                           END_REGION MQTT_COMMAND_SEND_PING
                         #MQTT_COMMAND_STATE_PING_RESP:
                           REGION WAIT_FOR_PING_RESP
                             //check watchdog status
                             IF #instTimerCommandWatchdog.Q THEN
                               #statEnableTimerCommandWatchdog := FALSE;
                               #statStatus := #ERR_MQTT_COMMAND_SEND_TIMEOUT; // Set correct status that identifies error clearly
                               #statSubfunctionStatus := #ERR_MQTT_COMMAND_SEND_TIMEOUT; // Status or return value of called FBs, FCs and system blocks
                               #statFBErrorState := #statFBState; // Set error state number for diagnostic 
                               #statErrorAutoCleared := TRUE;
                               #statMqttCommandState := #MQTT_COMMAND_STATE_NO_PROCESSING;
                             END_IF;
                             //Check PingRsp paket
                             CASE #tempMqttPingRspRcv OF
                               #NO_RESPONSE:  // Statement section case 1
                                 ;
                               #RESPONSE_GOOD:
                                 //disable watchdog
                                 #statEnableTimerCommandWatchdog := FALSE;
                                 //Go to no processing
                                 #statMqttCommandState := #MQTT_COMMAND_STATE_NO_PROCESSING;
                                 //set Status
                                 #statStatus := #STATUS_MQTT_CONNECTED;
                             END_CASE;
                           END_REGION MQTT_COMMAND_PING_RESP
                         ELSE  // Statement section ELSE
                           REGION ERROR_MULITPLE_INPUT
                             #statMqttCommandState := #MQTT_COMMAND_STATE_NO_PROCESSING; // reset back to idle
                             #statStatus := #ERR_MQTT_COMMAND_MULTIPLE_INPUT; // Set correct status that identifies error clearly
                             #statSubfunctionStatus := #ERR_MQTT_COMMAND_MULTIPLE_INPUT; // Status or return value of called FBs, FCs and system blocks
                             #statFBErrorState := #statFBState; // Set error state number for diagnostic 
                             #statErrorAutoCleared := TRUE;
                           END_REGION ERROR_MULITPLE_INPUT 
                       END_CASE;
                     END_REGION

                     REGION CHECK_PING_TIMER
                       //If no job is running check if keepalive experied
                       IF #statMqttCommandState = #MQTT_COMMAND_STATE_NO_PROCESSING
                         AND #instMqttKeepAliveTimer.Q THEN
                         //reset the timer
                         RESET_TIMER(#instMqttKeepAliveTimer);
                         //go to ping state
                         #statMqttCommandState := #MQTT_COMMAND_STATE_SEND_PING;
                       END_IF;
                     END_REGION CHECK_PING_TIMER

                     //Edge detection "publish / subscribe/unsubscribe" input
                     #statPublishOld := #tempPublish;
                     #statSubscribeOld := #tempSubscribe;
                     #statUnsubscribeOld := #tempUnsubscribe;

                     //Reset Done Bit
                     IF #statPublishOld = FALSE AND
                       #statSubscribeOld = FALSE AND
                       #statUnsubscribeOld = FALSE
                     THEN
                       #statDone := FALSE;
                     END_IF;

                   END_REGION CONNECTED

                 ELSE   // Undefined state in state machine reached
                   #statStatus := #ERR_UNDEFINED_STATE;
                   #statErrorUserCleared := TRUE;
               END_CASE;

             END_REGION MQTT_STATE_MACHINE
           END_IF;
         END_REGION FB_OPERATING_MONITOR_TCP

       #FB_STATE_TCP_RECONNECTING:
         REGION FB_STATE_TCP_RECONNECTING
           IF #tempTsendcStatus = #TSENDC_EST_OK THEN
             #statErrorAutoCleared := FALSE;
             //Monitor Connection
             #statFBState := #FB_STATE_OPERATING_MONITOR_TCP;
             // Begin MQTT Connection
             #statMqttConnectState := #MQTT_CONNECT_STATE_BUILD_PAKET;
           END_IF;
         END_REGION FB_STATE_TCP_RECONNECTING
       #FB_STATE_DISABLING: // Disabling active
         REGION DISABLING FB
           //  Disabling, e.g. closing connections, etc.
           // When disabling is complete the bit #statDisablingCompleted must be set
           // When MQTT is connected, send disconnect
           IF #statMqttConnectState = #MQTT_CONNECT_STATE_CONNECTED THEN
             IF #statTsendcReq = TRUE THEN
               //Interrupt any existing send jobs
               #statTsendcReq := FALSE;
             ELSE
               // INIT
               #statSendBufferPos := 0;
               //Build fixed Header
               //Message Type
               #statSendBuffer[#statSendBufferPos] := #MQTT_MSG_TYPE_DISCONNECT;
               #statSendBufferPos += 1;
               //Remaining Length (must be O)
               #statSendBuffer[#statSendBufferPos] := #REMAINIG_LEN_0;
               #statSendBufferPos += 1;
               //send request
               #statTsendcLen := #statSendBufferPos;
               #statTsendcReq := TRUE;
               #statMqttConnectState := #MQTT_CONNECT_STATE_DISCONNECTED;
             END_IF;
           ELSE
             //Disable TCP Connection
             #statTsendcReq := FALSE;
             #statTsendcEnable := FALSE;
             #statEnableTimerCommandWatchdog := TRUE;
           END_IF;
           // When TCP connection is closed
           IF #tempTsendcStatus = #TSENDC_DISCONNECTED THEN
             #statEnableTimerCommandWatchdog := FALSE;
             #statDisablingCompleted := TRUE;
           ELSIF #instTimerCommandWatchdog.Q THEN
             #statEnableTimerCommandWatchdog := FALSE;
             #statDisablingCompleted := TRUE;
           END_IF;
         END_REGION DISABLING FB
       ELSE // Undefined state in state machine reached
         #statStatus := #ERR_UNDEFINED_STATE;
         #statErrorUserCleared := TRUE;
     END_CASE;
   END_REGION STATE_MACHINE

   REGION OUTPUTS
     // Write outputs
     IF (#statDisablingCompleted = TRUE) THEN
       // Reset outputs if disabling completed
       #statValid := FALSE;
       #statBusy := FALSE;
       #statError := FALSE;
       #statDone := FALSE;
       #statErrorUserCleared := FALSE;
       #statErrorAutoCleared := FALSE;
       #statStatus := #STATUS_NO_CALL;
       // Reset application specific outputs
       #statRcvMsgStatus := #MSG_DECODE_STATUS_NO_NEW_MSG;
       #statRcvMsgDataLen := 0;
     ELSIF (#statErrorUserCleared = TRUE) AND (#statError = FALSE) THEN
       // Error can only be cleared by user; rising edge at enable input is needed to continue 
       #statValid := FALSE;
       #statBusy := FALSE;
       #statDone := FALSE;
       #statError := TRUE;
       // Write diagnostics
       #diagnostics.status := #statStatus;
       #diagnostics.subfunctionStatus := #statSubfunctionStatus;
       #diagnostics.stateNumber := #statFBErrorState;
       // execution aborted --> set state no processing
       #statTsendcEnable := FALSE; // Terminate Connection, no reason keep it up.
       #statFBState := #FB_STATE_NO_PROCESSING;
       #statMqttConnectState := #MQTT_CONNECT_STATE_NO_PROCESSING;
       #statMqttCommandState := #MQTT_COMMAND_STATE_NO_PROCESSING;
       #statRcvMsgDecodeState := #MSG_DECODE_STATE_NO_PROCESSING;

     ELSIF (#statErrorAutoCleared = TRUE) AND (#statError = FALSE) THEN
       // Error can be reset by FB automatically
       #statValid := FALSE;
       #statBusy := TRUE;
       #statError := TRUE;
       #statDone := FALSE;
       // Write diagnostics
       #diagnostics.status := #statStatus;
       #diagnostics.subfunctionStatus := #statSubfunctionStatus;
       #diagnostics.stateNumber := #statFBErrorState;
       // Handling of autocleared error
       CASE #statStatus OF
           //Just signal error and reset autocleared error afterwards.
         #ERR_MQTT_PAKET_ID_INVALID, #ERR_MQTT_SUBACK_FAILURE, #ERR_MQTT_CONNECT_TIMEOUT,
         #ERR_MQTT_COMMAND_SEND_TIMEOUT, #ERR_MQTT_COMMAND_MULTIPLE_INPUT, #ERR_CNT_EXCEEDS_ARRAY_DIMENSION,
         #ERR_MQTT_COMMAND_PUBLISH_TOPIC_INVALID, #ERR_QOS_INVALID, #ERR_MQTT_COMMAND_SUBSCRIBE_TOPIC_INVALID:
           #statErrorAutoCleared := FALSE;

         ELSE  // Statement section ELSE
           ;
       END_CASE;

     ELSIF (#statErrorAutoCleared = FALSE) AND (#statErrorUserCleared = FALSE) AND (#statError = TRUE) THEN
       // If autocleared error is acknowledged
       #statValid := TRUE;
       #statBusy := TRUE;
       #statError := FALSE;
       #statDone := FALSE;
       //   this line  more detailed status information is used instead of "#STATUS_SUBSEQUENT_CALL"
       CASE #statStatus OF
         #ERR_TCP_RECONNECTING, #ERR_MQTT_CONNECT_TIMEOUT:  // Reconnecting ok, start Mqtt reconnnect
           //set status
           #statStatus := #STATUS_MQTT_CONNECTING;
           //in the following status codes status stays connected. 
         #ERR_MQTT_PAKET_ID_INVALID, #ERR_MQTT_SUBACK_FAILURE, #ERR_MQTT_COMMAND_SEND_TIMEOUT,
         #ERR_MQTT_COMMAND_MULTIPLE_INPUT, #ERR_CNT_EXCEEDS_ARRAY_DIMENSION, #ERR_MQTT_COMMAND_PUBLISH_TOPIC_INVALID,
         #ERR_QOS_INVALID, #ERR_MQTT_COMMAND_SUBSCRIBE_TOPIC_INVALID:
           #statStatus := #STATUS_MQTT_CONNECTED;
         ELSE  // Statement section ELSE
           ;
       END_CASE;
     END_IF;

     // Write static values to outputs
     #valid := #statValid;
     #busy := #statBusy;
     #error := #statError;
     #status := #statStatus;
     //block sets ENO automatically:
     //ENO := TRUE;
     //Write application specific static values to outputs
     #done := #statDone;
     #receivedMsgStatus := #statRcvMsgStatus;
     #receivedMsgDataLen := #statRcvMsgDataLen;
   END_REGION OUTPUTS
END_FUNCTION_BLOCK

// folder: LMQTT/Utilities

FUNCTION "LMQTT_ConvertToUtf8" : Void   // FC6, SCL
TITLE = LMQTT_ConvertToUtf8
{ S7_Optimized_Access := 'TRUE' }
AUTHOR : SIEMENS
FAMILY : LMQTT
VERSION : 1.0
// Function to convert a WCHAR to a UTF-8 conformant byte sequence
   VAR_INPUT
      character : WChar;   // Character that shall be converted to UTF-8
   END_VAR
   VAR_OUTPUT
      convertedUtf8 : DWord;   // UTF-8 conformant byte sequence. B0 stores first Byte, B1 second and B2 third Byte. B3 is not used
      bytesUsed : USInt;   // Amount of Bytes converted. Ranges from 1 to 3.
      error : Bool;   // TRUE: An error occurred during the execution of the FC
      status : Word;   // 16#0000 - 16#7FFF: Status of the FC, 16#8000 - 16#FFFF: Error identification
   END_VAR
   VAR_TEMP
      tempStatus : Word;   // temp value for output 'status'
      tempConvertedUtf8 : DWord;   // temp value for output 'convertedUtf8'
      tempBytesUsed : USInt;   // temp value for output 'bytesUsed'
      tempCharacter : WChar;   // temp value for input 'character'
   END_VAR
   // Ret_Val : No return for this FC - see error and status output
   VAR CONSTANT
      STATUS_NO_ERROR : Word := 16#0000;   // no error status
      STATUS_EXECUTION_FINISHED : Word := 16#0000;   // Execution finished without errors
      ERR_UNDEFINED : Word := 16#8000;   // Error due to an undefined case
      USINT_NULL : USInt := 0;   // Init value with 0
      DWORD_NULL : DWord := 16#0000_0000;   // Init value with 0
      EMPTY_WCHAR : WChar := WCHAR#' ';   // Empty WChar for comparison
      BELOW_7F : Word := 16#007F;   // Upper limit for character if only one Byte used
      BELOW_7FF : Word := 16#07FF;   // Upper limit for character if two Byte used
      BELOW_MAX_FFFF : Word := 16#FFFF;   // Upper limit for character if three Byte used
      BYTE_3F : Byte := 16#3F;   // Conversion Value
      BYTE_80 : Byte := 16#80;   // Conversion Value
      BYTE_C0 : Byte := 16#C0;   // Conversion Value
      BYTE_E0 : Byte := 16#E0;   // Conversion Value
      USINT_ONE : USInt := 1;   // Const Value to assign amount of bytes used
      USINT_TWO : USInt := 2;   // Const Value to assign amount of bytes used
      USINT_THREE : USInt := 3;   // Const Value to assign amount of bytes used
   END_VAR
BEGIN
   REGION BLOCK INFO HEADER
       //=============================================================================
       // SIEMENS AG
       // (c)Copyright 2020
       //-----------------------------------------------------------------------------
       // Library:       LMQTT
       // Tested with:   CPU 1516-3 PN/DP V2.8
       // Engineering:   TIA Portal V16
       // Restrictions:  --
       // Requirements:  --
       // Functionality: Converts a single WChar Character to a valid UTF-8 encoded byte sequence and saves this to a DWord.
       //                The amount of bytes saved is stored in bytesUsed Output.
       //-----------------------------------------------------------------------------
       // Change log table:
       // Version    Date         Expert in charge         Changes applied
       // 03.00.00   01.10.2020   Siemens Online Support   First released version
       //=============================================================================
   END_REGION

   REGION INITIALISATION  
       // Initialize functionality: reset of variables, diagnostics, etc.
       #tempConvertedUtf8 := #DWORD_NULL;
       #tempBytesUsed := #USINT_NULL;
       #tempStatus := #STATUS_NO_ERROR;
       //assign temp value from input:
        #tempCharacter := #character;

   END_REGION

   REGION PROGRAM LOGIC
       // Use this region for application specific code
       IF #tempCharacter = #EMPTY_WCHAR THEN
           //will be only 1 byte occupied
           #tempConvertedUtf8 := WCHAR_TO_DWORD(#tempCharacter);
           #tempBytesUsed := #USINT_ONE;
       ELSIF (WCHAR_TO_WORD(#tempCharacter) <= (#BELOW_7F)) THEN
           //will be only 1 byte occupied
           #tempConvertedUtf8 := WCHAR_TO_DWORD(#tempCharacter);
           #tempBytesUsed := #USINT_ONE;
       ELSIF (WCHAR_TO_WORD(#tempCharacter) <= (#BELOW_7FF)) THEN
           //will be 2 byte occupied
           #tempConvertedUtf8.%B1 := (WCHAR_TO_BYTE(#tempCharacter) AND #BYTE_3F) OR #BYTE_80;
           #tempConvertedUtf8.%B0 := WORD_TO_BYTE(SHR(IN := WCHAR_TO_WORD(#tempCharacter), N := 6)) OR #BYTE_C0;
           #tempBytesUsed := #USINT_TWO;
       ELSIF (WCHAR_TO_WORD(#tempCharacter) <= (#BELOW_MAX_FFFF)) THEN
           //will be 3 byte occupied
           #tempConvertedUtf8.%B2 := (WCHAR_TO_BYTE(#tempCharacter) AND #BYTE_3F) OR #BYTE_80;
           #tempConvertedUtf8.%B1 := (WORD_TO_BYTE(SHR(IN := WCHAR_TO_WORD(#tempCharacter), N := 6)) AND #BYTE_3F) OR #BYTE_80;
           #tempConvertedUtf8.%B0 := WORD_TO_BYTE(SHR(IN := WCHAR_TO_WORD(#tempCharacter), N := 12)) OR #BYTE_E0;
           #tempBytesUsed := #USINT_THREE;
       END_IF;
   END_REGION

   REGION OUTPUTS
       // Write application specific temp values to outputs
       #bytesUsed := #tempBytesUsed;
       #convertedUtf8 := #tempConvertedUtf8;
       // Write error and status
       #error := #tempStatus.%X15;
       #status := #tempStatus;
       // ENO mechanism is not used --> ENO := TRUE;
       ENO := TRUE;
   END_REGION
END_FUNCTION

// ===== library types =====

FUNCTION_BLOCK "LMqtt_Publisher"   // FB2, SCL
{ S7_Optimized_Access := 'TRUE' }
VERSION : 0.1
   VAR_INPUT
      enable : Bool;
      publish : Bool;
      tcpConnParam : "typeTcpConnParam";
      mqttParam : "typeMqttParam";
   END_VAR
   VAR_OUTPUT
      tcpEstablished : Bool;
      mqttEstablished : Bool;
      published : Bool;
      busy : Bool;
      error : Bool;
      status : DWord;
      statusID : Int;
   END_VAR
   VAR
      statTcpConnParam : TCON_IP_v4;
      instTcpConnect : TCON;
      instTcpSend : TSEND;
      instTcpRCV : TRCV;
      instTcpDisconnect : TDISCON;
      instWatchDog : TON_TIME;
      instKeepAlive : TON_TIME;
      statStateMQTT : Int;
      statStateMQTTinternal : Int;
      statStateTCP : Int;
      statLastState : Int;
      statConnectLenght : Int;
      statCorrectOffset : Int;
      statSendLenght : Int;
      statConnectEncodedLenght : Int;
      statConnectLenghtOffset : Int;
      statKeepAliveTime : Time;
      statI : Int;
      statPacketID : Word;
      statPacketIDAck : Word;
      statRcvLen : UDInt;
      statPublishOld : Bool;
      statReConnect : Bool;
      statEnableOld : Bool;
      statMqttResetOld : Bool;
      statTriggerWatchDog : Bool;
      statTriggerKeepAlive : Bool;
      statNewDataRcv : Bool;
      statKeepAliveOff : Bool;
      statSendBuffer : Array[1..1000] of Byte;
      statRcvBuffer : Array[1..200] of Byte;
   END_VAR
   VAR_TEMP
      tempStringToChar : Array[0..255] of Char;
      tempCountChars : UInt;
      tempLenght : Word;
   END_VAR
   VAR CONSTANT
      TCP_PARAM : Int := 1;
      TCP_DISCONNECT : Int := -1;
      TCP_ERROR : Int := -2;
      TCP_CONNECTED : Int := 3;
      TCP_CONNECTING : Int := 2;
      MQTT_CONNECT_FLAG_CHECK : Int := 10;
      MQTT_CONNECT : Int := 11;
      MQTT_PUBLISH : Int := 13;
      MQTT_DISCONNECT : Int := 15;
      MQTT_CONNACK : Int := 12;
      MQTT_PUBACK : Int := 14;
      MQTT_PING : Int := 17;
      MQTT_PINGRESP : Int := 18;
      MQTT_PUBREL : Int := 19;
      MQTT_PUBCOMP : Int := 20;
      MQTT_IDLE : Int;
      MQTT_CONNECTED : Int := 16;
      MQTT_DISCONNECTED : Int := -11;
      MQTT_ERROR : Int := -12;
      IDLE : Int;
      TIME_MONITORING : Int := 20;
      WATCHDOG_TIME : Time := t#30s;
      MQTT_MSG_TYPE_CONNACK : Int := 32;
      MQTT_MSG_TYPE_DISCONNECT : Int := 224;
      MQTT_MSG_TYPE_PUBACK : Int := 64;
      MQTT_MSG_TYPE_PUBREC : Int := 80;
      MQTT_MSG_TYPE_PUBCOM : Int := 112;
      MQTT_MSG_TYPE_PING : Int := 192;
      MQTT_MSG_TYPE_PINGRESP : Int := 208;
      MQTT_CONNACK_ACCEPTED : Int;
      MQTT_PORT : Word := 16#22B3;
      MQTT_PROTOCOL_NAME : String := 'MQTT';
      MQTT_ERROR_WILL_FLAG : Word := 16#80F0;
      MQTT_ERROR_QOS_FLAG : Word := 16#80F1;
      MQTT_ERROR_PACKETID : Word := 16#80F2;
      MQTT_ERROR_KEEPALIVE : Word := 16#80F3;
   END_VAR
   // statTcpConnParam.ActiveEstablished := true;
BEGIN
   //=============================================================================
   //SIEMENES AG
   //(c)Copyright 2016 All Rights Reserved
   //-----------------------------------------------------------------------------
   //Library:       (that the source is dedicated to)
   //Tested with:   (target system with FW Version)
   //Engineering:   TIA Portal V15
   //Restrictions:  (OB types, etc.)
   //Requirements:  (hardware, technological package, memory needed, etc.)
   //Functionality: MQTT
   //-----------------------------------------------------------------------------
   //Change log table:
   //Version  Date       Expert in charge Changes applied
   //01.00.00 dd.mm.yyyy (name of expert) First released version
   //=============================================================================
   //Establish TCP Connection to be ready for MQTT

   IF #enable
       AND NOT #statEnableOld
   THEN
       #statStateTCP := #TCP_PARAM;
       #statStateMQTT := #MQTT_DISCONNECTED;
       #instWatchDog.IN := false;
       #statPublishOld := #publish;
       #error := 0;
       #status := 0;
       #statusID := 0;
   END_IF;

   IF NOT #enable
       AND #statEnableOld
   THEN
       IF #statStateTCP = #TCP_CONNECTED AND
           #statStateMQTT = #MQTT_DISCONNECTED
       THEN
           #statStateTCP := #TCP_DISCONNECT;
       END_IF;
       IF #statStateTCP = #TCP_CONNECTED AND
           #statStateMQTT <> #MQTT_DISCONNECTED
       THEN
           #statStateMQTT := #MQTT_DISCONNECT;
       END_IF;
       IF #statStateTCP = #TCP_CONNECTING
           OR  #statStateTCP = #IDLE
       THEN

           #statStateMQTT := #MQTT_DISCONNECTED;
           #statStateTCP := #IDLE;
       END_IF;
   END_IF;

    #instWatchDog(IN := #statTriggerWatchDog,PT := #WATCHDOG_TIME);

   REGION State maschine TCP
       CASE #statStateTCP OF
           #IDLE:
               IF NOT #error
               THEN
                   #status := 0;
                   #statusID := 0;

               END_IF;
               #statTcpConnParam.ID := #tcpConnParam.connectionID;
               #instTcpDisconnect(ID := #statTcpConnParam.ID);
               #instTcpConnect(ID := #statTcpConnParam.ID,
                               CONNECT := #statTcpConnParam);
               #published := 0;
               #busy := false;
               #mqttEstablished := false;
               #statMqttResetOld := 0;
               #tcpEstablished := false;
               #statStateMQTT := #MQTT_DISCONNECTED;
               #statStateMQTTinternal := #IDLE;
               #statTriggerWatchDog := false;
               #statTriggerKeepAlive := 0;
               IF #statLastState=#TCP_DISCONNECT
               THEN
                   #error := 0;
                   END_IF;
           #TCP_CONNECTED:
               ;
               //Check TCP Connection
               IF #instTcpRCV.STATUS > w#16#80C0
               THEN
                   #statStateTCP := #TCP_ERROR;
                   #statusID := #TCP_CONNECTED;
               END_IF;
               #statLastState := #TCP_CONNECTED;
           #TCP_PARAM:
               #statTcpConnParam.InterfaceId := #tcpConnParam.hwIdentifier;
               #statTcpConnParam.ID := #tcpConnParam.connectionID;
               #statTcpConnParam.LocalPort := #tcpConnParam.localPort;
               #statTcpConnParam.RemotePort := #tcpConnParam.mqttPort;
               #statTcpConnParam.ActiveEstablished := true;
               #statTcpConnParam.RemoteAddress.ADDR[1] := #tcpConnParam.ipAdressBroker[0];
               #statTcpConnParam.RemoteAddress.ADDR[2] := #tcpConnParam.ipAdressBroker[1];
               #statTcpConnParam.RemoteAddress.ADDR[3] := #tcpConnParam.ipAdressBroker[2];
               #statTcpConnParam.RemoteAddress.ADDR[4] := #tcpConnParam.ipAdressBroker[3];

             #statStateTCP := #TCP_CONNECTING;
           #TCP_CONNECTING:
               REGION TCP Connect
                   #statTriggerWatchDog := true;
                   #instTcpConnect.REQ := NOT #instTcpConnect.REQ XOR #instTcpConnect.BUSY;
                   #instTcpConnect(ID := #statTcpConnParam.ID,
                                   CONNECT := #statTcpConnParam);

                   IF (#instTcpConnect.DONE)
                       AND (#instTcpConnect.BUSY = 0)
                       AND (#instTcpConnect.REQ)
                   THEN
                       #instTcpConnect.REQ := false;
                       #tcpEstablished := true;
                       #statStateTCP := #TCP_CONNECTED;
                       #statTriggerWatchDog := false;
                   ELSIF (#instTcpConnect.ERROR)
                   THEN
                       #statusID := #TCP_CONNECTING;
                       #instTcpConnect.REQ := false;
                       #statStateTCP := #TCP_ERROR;
                   END_IF;
               END_REGION

           #TCP_DISCONNECT:
               REGION TCP Disconnect
                   #instTcpDisconnect.REQ := NOT #instTcpDisconnect.REQ XOR #instTcpDisconnect.BUSY;
                   #statTriggerWatchDog := false;
                   #instTcpDisconnect(ID := #statTcpConnParam.ID);

                   IF (#instTcpDisconnect.DONE)
                   THEN
                       //Done with success
                       #instTcpDisconnect.REQ := false;
                       #statLastState := #TCP_DISCONNECT;
                       #statStateTCP := #IDLE;
                   ELSIF (#instTcpDisconnect.ERROR)
                   THEN
                       #statusID := #TCP_DISCONNECT;
                       #instTcpDisconnect.REQ := false;
                       #statStateTCP := #TCP_ERROR;
                   END_IF;
               END_REGION
               ;
           #TCP_ERROR:
               REGION Errorhandling
                   #error := true;
                   #statStateMQTT := #MQTT_DISCONNECTED;
                   #statStateMQTTinternal := #IDLE;
                   #tcpEstablished := false;
                   #mqttEstablished := false;
                   #published := false;
                   #statTriggerWatchDog := false;
                   #instTcpConnect.REQ := false;
                       CASE #statusID OF
                           #TCP_CONNECTING:
                               #statStateTCP := #IDLE;
                               #status := #instTcpConnect.STATUS;
                           #TCP_CONNECTED:
                               #statStateTCP := #TCP_DISCONNECT;
                               #status := #instTcpRCV.STATUS;
                           #TCP_DISCONNECT:
                               //pointless for a retry at TDISCON
                               #statStateTCP := #IDLE;
                               #status := #instTcpDisconnect.STATUS;
                           #TIME_MONITORING:
                               IF (#statLastState = #TCP_CONNECTED)
                               THEN
                                   #statStateTCP := #TCP_DISCONNECT;
                                   #status := #instTcpRCV.STATUS;
                               ELSE
                                   #statStateTCP := #IDLE;
                                   #status := #instTcpConnect.STATUS;
                               END_IF;
                           ELSE
                               ;
                       END_CASE;
               END_REGION
               ;
           ELSE
               ;
       END_CASE;
   END_REGION
   #statEnableOld := #enable;
   REGION WatchDog
       IF #instWatchDog.Q = true
       THEN
           #statStateTCP := #TCP_ERROR;
           #statusID := #TIME_MONITORING;
       END_IF;
   END_REGION

   REGION OUC blocks

       #instTcpSend(ID:=#statTcpConnParam.ID,
                     DATA:=#statSendBuffer);
        #instTcpRCV(EN_R:=true,
                    ID:=#statTcpConnParam.ID,
                   LEN:=0,
                   ADHOC:=1,
                   RCVD_LEN=>#statRcvLen,
                   DATA:=#statRcvBuffer);
       IF #instTcpRCV.RCVD_LEN > 0 THEN
           #statNewDataRcv := 1;
       END_IF;

   END_REGION

   //Bring Statemachine in a definded state, if TCP Connection breaks
   IF #statStateMQTT > 0 AND
       #statStateTCP <> #TCP_CONNECTED
   THEN
       #statStateMQTT := #MQTT_DISCONNECTED;
       #instTcpSend.REQ := 0;
   END_IF;

   //MQTT makes no sense without an established TCP
   IF NOT (#statStateTCP = #TCP_CONNECTED)
   THEN
       RETURN;
   END_IF;




    #instKeepAlive(IN := #statTriggerKeepAlive,
                   PT := #statKeepAliveTime);
       CASE #statStateMQTT OF
           #MQTT_DISCONNECTED:
               #mqttEstablished := false;
               #statPublishOld := #publish;
               #statStateMQTT := #MQTT_CONNECT_FLAG_CHECK;
               #statStateMQTTinternal := #IDLE;
               #statTriggerKeepAlive := 0;
               #statKeepAliveOff := false;
               #statPacketID := #mqttParam.packetIdentifier;

           #MQTT_CONNECT_FLAG_CHECK:
               #busy := 1;
               //validate flags
               IF #mqttParam.connectFlag.willRetain
                   AND NOT #mqttParam.connectFlag.will
               THEN
                   #statStateMQTT := #MQTT_ERROR;
                   #statusID := #MQTT_CONNECT_FLAG_CHECK;
                   #status := #MQTT_ERROR_WILL_FLAG;
               ELSE
                   IF NOT #mqttParam.connectFlag.will
                       AND (#mqttParam.connectFlag.willQoS_1 OR #mqttParam.connectFlag.willQoS_2)
                   THEN
                       #statStateMQTT := #MQTT_ERROR;
                       #statusID := #MQTT_CONNECT_FLAG_CHECK;
                       #status := #MQTT_ERROR_QOS_FLAG;
                   ELSE
                       IF (#mqttParam.connectFlag.willQoS_1
                           AND #mqttParam.connectFlag.willQoS_2)
                       THEN
                           #statStateMQTT := #MQTT_ERROR;
                           #statusID := #MQTT_CONNECT_FLAG_CHECK;
                           #status := #MQTT_ERROR_QOS_FLAG;
                       ELSE;
                        #statStateMQTT := #MQTT_CONNECT;
                       END_IF;
                   END_IF;

               END_IF;
               IF (WORD_TO_INT(#mqttParam.keepAlive) = 0)
               THEN
                   #statKeepAliveOff := true;
               END_IF;
               IF (WORD_TO_INT(#mqttParam.keepAlive) < 2)
                   AND
                   (WORD_TO_INT(#mqttParam.keepAlive) > 0)
               THEN
                   #statStateMQTT := #MQTT_ERROR;
                   #statusID := #MQTT_CONNECT_FLAG_CHECK;
                   #status := #MQTT_ERROR_KEEPALIVE;
               END_IF;
               IF (WORD_TO_INT(#mqttParam.keepAlive) > 2)
               THEN
                   #statKeepAliveOff := false;
               END_IF;
           #MQTT_CONNECT:
                REGION MQTT Connect

                   //Calculate Remaining Lenght
                   #statConnectLenght := 10 + LEN(IN := #mqttParam.clientIdentifier) + 2;
                   IF #mqttParam.connectFlag.userName
                   THEN
                       #statConnectLenght := #statConnectLenght + LEN(IN := #mqttParam.userName) + 2;
                   END_IF;
                   IF #mqttParam.connectFlag.password
                   THEN
                       #statConnectLenght := #statConnectLenght + LEN(IN := #mqttParam.password) + 2;
                   END_IF;
                   IF #mqttParam.connectFlag.will
                   THEN
                       #statConnectLenght := #statConnectLenght + LEN(IN := #mqttParam.willMessage) + LEN(IN := #mqttParam.willTopic) + 4;
                   END_IF;
                   #statConnectLenghtOffset := 0;
                   //Build Telegram
                   //Fixed Header
                   #statSendBuffer[1] := 16#10;

                   #statSendLenght :=#statConnectLenght;
                   WHILE (#statConnectLenght > 0)
                   DO
                       #statConnectEncodedLenght := #statConnectLenght MOD 128;
                       #statConnectLenght := #statConnectLenght / 128;
                       // if there are more data to encode, set the top bit of this byte
                       IF #statConnectLenght > 0
                       THEN
                           #statConnectEncodedLenght := #statConnectEncodedLenght OR 128;
                           #statSendBuffer[2 + #statConnectLenghtOffset] := INT_TO_BYTE(#statConnectEncodedLenght);
                           #statConnectLenghtOffset := #statConnectLenghtOffset + 1;
                       ELSE
                           #statSendBuffer[2 + #statConnectLenghtOffset] := INT_TO_BYTE(#statConnectEncodedLenght);
                       END_IF;
                   END_WHILE;
                   #statSendLenght := #statSendLenght + #statConnectLenghtOffset;
                   //Variable Header
                   //Protocol name
                   #statSendBuffer[3 + #statConnectLenghtOffset] := 0;
                   #statSendBuffer[4 + #statConnectLenghtOffset] := 4;
                   #statSendBuffer[5 + #statConnectLenghtOffset] := 'M';
                   #statSendBuffer[6 + #statConnectLenghtOffset] := 'Q';
                   #statSendBuffer[7 + #statConnectLenghtOffset] := 'T';
                   #statSendBuffer[8 + #statConnectLenghtOffset] := 'T';
                   //Protocol Level
                   #statSendBuffer[9 + #statConnectLenghtOffset] := 4;
                   //Connect Flags
                   #statSendBuffer[10 + #statConnectLenghtOffset].%X0 := 0;
                   #statSendBuffer[10 + #statConnectLenghtOffset].%X1 := #mqttParam.connectFlag.cleanSession;
                   #statSendBuffer[10 + #statConnectLenghtOffset].%X2 := #mqttParam.connectFlag.will;
                   #statSendBuffer[10 + #statConnectLenghtOffset].%X3 := #mqttParam.connectFlag.willQoS_1;
                   #statSendBuffer[10 + #statConnectLenghtOffset].%X4 := #mqttParam.connectFlag.willQoS_2;
                   #statSendBuffer[10 + #statConnectLenghtOffset].%X5 := #mqttParam.connectFlag.willRetain;
                   #statSendBuffer[10 + #statConnectLenghtOffset].%X6 := #mqttParam.connectFlag.password;
                   #statSendBuffer[10 + #statConnectLenghtOffset].%X7 := #mqttParam.connectFlag.userName;
                   //Keep Alive in sec
                  #statSendBuffer[11 + #statConnectLenghtOffset] := #mqttParam.keepAlive.%B1;
                  #statSendBuffer[12 + #statConnectLenghtOffset] := #mqttParam.keepAlive.%B0;
                   //Payload
                   //ClientIdentifier
                   #tempLenght := INT_TO_WORD(LEN(IN := #mqttParam.clientIdentifier));
                   #statSendBuffer[13 + #statConnectLenghtOffset] := #tempLenght.%B1;
                   #statSendBuffer[14 + #statConnectLenghtOffset] := #tempLenght.%B0;
                   Strg_TO_Chars(Strg := #mqttParam.clientIdentifier,
                                 pChars := 0,
                                 Cnt => #tempCountChars,
                                 Chars := #tempStringToChar);
                   FOR #statI := 0 TO UINT_TO_INT(#tempCountChars - 1) DO
                       #statSendBuffer[15 + #statConnectLenghtOffset + #statI] := #tempStringToChar[#statI];
                   END_FOR;
                   #statConnectLenghtOffset := #statConnectLenghtOffset + #statI;
                   //WillTopic and WillMessage
                   IF #mqttParam.connectFlag.will THEN
                       #statCorrectOffset := 0;
                       #tempLenght:=INT_TO_WORD(LEN(IN := #mqttParam.willTopic));
                       #statSendBuffer[15 + #statConnectLenghtOffset] := #tempLenght.%B1;
                       #statSendBuffer[16 + #statConnectLenghtOffset] := #tempLenght.%B0;
                       Strg_TO_Chars(Strg := #mqttParam.willTopic,
                                     pChars := 0,
                                     Cnt => #tempCountChars,
                                     Chars := #tempStringToChar);
                       FOR #statI := 0 TO UINT_TO_INT(#tempCountChars - 1) DO
                           #statSendBuffer[17 + #statConnectLenghtOffset + #statI] := #tempStringToChar[#statI];
                       END_FOR;
                       #statConnectLenghtOffset := #statConnectLenghtOffset + #statI;

                       #tempLenght:=INT_TO_WORD(LEN(IN := #mqttParam.willMessage));
                       #statSendBuffer[17 + #statConnectLenghtOffset] := #tempLenght.%B1;
                       #statSendBuffer[18 + #statConnectLenghtOffset] := #tempLenght.%B0;
                       Strg_TO_Chars(Strg := #mqttParam.willMessage,
                                     pChars := 0,
                                     Cnt => #tempCountChars,
                                     Chars := #tempStringToChar);
                       FOR #statI := 0 TO UINT_TO_INT(#tempCountChars - 1) DO
                           #statSendBuffer[19 + #statConnectLenghtOffset + #statI] := #tempStringToChar[#statI];
                       END_FOR;
                       #statConnectLenghtOffset := #statConnectLenghtOffset + #statI;
                   ELSE
                       #statCorrectOffset := 4;
                   END_IF;
                   //UserName
                   IF #mqttParam.connectFlag.userName THEN
                       #tempLenght := INT_TO_WORD(LEN(IN := #mqttParam.userName));
                       #statSendBuffer[19 + #statConnectLenghtOffset - #statCorrectOffset] := #tempLenght.%B1;
                       #statSendBuffer[20 + #statConnectLenghtOffset - #statCorrectOffset] := #tempLenght.%B0;
                       Strg_TO_Chars(Strg := #mqttParam.userName,
                                     pChars := 0,
                                     Cnt => #tempCountChars,
                                     Chars := #tempStringToChar);
                       FOR #statI := 0 TO UINT_TO_INT(#tempCountChars - 1) DO
                           #statSendBuffer[21 + #statConnectLenghtOffset + #statI-#statCorrectOffset] := #tempStringToChar[#statI];
                       END_FOR;
                       #statConnectLenghtOffset := #statConnectLenghtOffset + #statI;
                   END_IF;
                   //Password
                   IF #mqttParam.connectFlag.password THEN
                       #tempLenght := INT_TO_WORD(LEN(IN := #mqttParam.password));
                       #statSendBuffer[21 + #statConnectLenghtOffset - #statCorrectOffset] := #tempLenght.%B1;
                       #statSendBuffer[22 + #statConnectLenghtOffset - #statCorrectOffset] := #tempLenght.%B0;
                       Strg_TO_Chars(Strg := #mqttParam.password,
                                     pChars := 0,
                                     Cnt => #tempCountChars,
                                     Chars := #tempStringToChar);
                       FOR #statI := 0 TO UINT_TO_INT(#tempCountChars - 1) DO
                           #statSendBuffer[23 + #statConnectLenghtOffset + #statI-#statCorrectOffset] := #tempStringToChar[#statI];
                       END_FOR;
                       #statConnectLenghtOffset := #statConnectLenghtOffset + #statI;
                   END_IF;

            #instTcpSend.REQ := true;
             #instTcpSend.LEN := INT_TO_UDINT(#statSendLenght + 2);

                   IF ((#instTcpSend.DONE)
                       AND (#instTcpSend.BUSY = 0))
                   THEN
                       #instTcpSend.REQ := false;
                       #statStateMQTT := #MQTT_CONNACK;
                       //Delete Send Buffer
                       FOR #statI := 1 TO (#statSendLenght + 2) DO
                           #statSendBuffer[#statI] := 0;
                       END_FOR;
                   ELSIF #instTcpSend.ERROR
                   THEN
                       #statusID := #MQTT_CONNECT;
                       #instTcpSend.REQ := false;
                       #statStateMQTT := #MQTT_ERROR;

                   END_IF;

               END_REGION
               ;
           #MQTT_CONNACK:
               IF #statNewDataRcv THEN

                   IF ((#statRcvBuffer[1] AND b#16#f0) = #MQTT_MSG_TYPE_CONNACK)
                       AND
                       (#statRcvBuffer[4] = #MQTT_CONNACK_ACCEPTED)
                   THEN
                       #statStateMQTT := #MQTT_CONNECTED;
                       #mqttEstablished := true;
                       #busy := false;
                       #statStateMQTTinternal := #IDLE;
                       //start Keep Alive Timer
                       //KeepAliveTImer is set to (Keep Alive (in s) - 2s)
                       #statKeepAliveTime := UINT_TO_TIME((WORD_TO_UINT(#mqttParam.keepAlive) * 1000 - 2000));
                       IF NOT #statKeepAliveOff
                       THEN
                           #statTriggerKeepAlive := true;
                       END_IF;
                       #statNewDataRcv := 0;
                   ELSE
                       #statStateMQTT := #MQTT_ERROR;
                       #statusID := #MQTT_CONNACK;
                   END_IF;
               END_IF;
           #MQTT_CONNECTED:
               IF #publish
                   AND NOT #statPublishOld
                   AND (#statStateMQTTinternal=#IDLE)
               THEN
                   #statStateMQTTinternal := #MQTT_PUBLISH;
                   #published := 0;
                   #error := 0;
                  #statTriggerKeepAlive := false;
                   #statPacketID := #statPacketID + 1;
               END_IF;
               #statPublishOld := #publish;

                IF (#instKeepAlive.Q)
                    AND (#statStateMQTTinternal = #IDLE)
                    AND (NOT #statKeepAliveOff)
                THEN
                    #statStateMQTTinternal := #MQTT_PING;
                    #statTriggerKeepAlive := false;
                END_IF;
                CASE #statStateMQTTinternal OF
                    #IDLE:
                        #published := 0;
                        ;
                    #MQTT_PUBLISH:
                        ;
                        #busy := true;
                        #statConnectLenghtOffset := 0;
                        #statConnectLenght := LEN(IN := #mqttParam.topic) + LEN(IN := #mqttParam.message) + 2;
                        #statSendBuffer[1] := 16#30;
                        #statSendBuffer[1].%X0 := #mqttParam.publishFlag.retain;
                        #statSendBuffer[1].%X3 := false;
                        CASE #mqttParam.publishFlag.qualityOfService OF
                            0:
                                #statSendBuffer[1].%X1 := 0;
                                #statSendBuffer[1].%X2 := 0;
                            1:
                                #statSendBuffer[1].%X1 := 1;
                                #statSendBuffer[1].%X2 := 0;
                                //2 Byte Packet Identifiert added
                                #statConnectLenght := #statConnectLenght + 2;
                            2:
                                #statSendBuffer[1].%X1 := 0;
                                #statSendBuffer[1].%X2 := 1;
                                //2 Byte Packet Identifiert added
                                #statConnectLenght := #statConnectLenght + 2;
                            ELSE:
                                ;
                                #statStateMQTT := #MQTT_ERROR;
                                #statusID := #MQTT_PUBLISH;
                        END_CASE;
                        #statSendLenght := #statConnectLenght;
                        WHILE (#statConnectLenght > 0)
                        DO
                            #statConnectEncodedLenght := #statConnectLenght MOD 128;
                            #statConnectLenght := #statConnectLenght / 128;
                            // if there are more data to encode, set the top bit of this byte
                            IF #statConnectLenght > 0
                            THEN
                                #statConnectEncodedLenght := #statConnectEncodedLenght OR 128;
                                #statSendBuffer[2 + #statConnectLenghtOffset] := INT_TO_BYTE(#statConnectEncodedLenght);
                                #statConnectLenghtOffset := #statConnectLenghtOffset + 1;
                            ELSE
                                #statSendBuffer[2 + #statConnectLenghtOffset] := INT_TO_BYTE(#statConnectEncodedLenght);
                            END_IF;
                        END_WHILE;
                        #statSendLenght := #statSendLenght + #statConnectLenghtOffset;
                        //Variable Header
                        #tempLenght := INT_TO_WORD(LEN(IN := #mqttParam.topic));
                        #statSendBuffer[3 + #statConnectLenghtOffset] := #tempLenght.%B1;
                        #statSendBuffer[4 + #statConnectLenghtOffset] := #tempLenght.%B0;
                        Strg_TO_Chars(Strg := #mqttParam.topic,
                                      pChars := 0,
                                      Cnt => #tempCountChars,
                                      Chars := #tempStringToChar);
                        FOR #statI := 0 TO UINT_TO_INT(#tempCountChars - 1) DO
                            #statSendBuffer[5 + #statConnectLenghtOffset + #statI] := #tempStringToChar[#statI];
                        END_FOR;
                        #statConnectLenghtOffset := #statConnectLenghtOffset + #statI;
                        IF (#mqttParam.publishFlag.qualityOfService > 0)
                        THEN

                            #statSendBuffer[5 + #statConnectLenghtOffset] := #statPacketID.%B1;
                            #statSendBuffer[6 + #statConnectLenghtOffset] := #statPacketID.%B0;
                            //Payload
                            Strg_TO_Chars(Strg := #mqttParam.message,
                                          pChars := 0,
                                          Cnt => #tempCountChars,
                                          Chars := #tempStringToChar);
                            FOR #statI := 0 TO UINT_TO_INT(#tempCountChars - 1) DO
                                #statSendBuffer[7 + #statConnectLenghtOffset + #statI] := #tempStringToChar[#statI];
                            END_FOR;
                            #instTcpSend.LEN := INT_TO_UDINT(#statSendLenght + 2);
                        ELSE
                            Strg_TO_Chars(Strg := #mqttParam.message,
                                          pChars := 0,
                                          Cnt => #tempCountChars,
                                          Chars := #tempStringToChar);
                            FOR #statI := 0 TO UINT_TO_INT(#tempCountChars - 1) DO
                                #statSendBuffer[5 + #statConnectLenghtOffset + #statI] := #tempStringToChar[#statI];
                            END_FOR;
                            #instTcpSend.LEN := INT_TO_UDINT(#statSendLenght + 2);
                        END_IF;

                        #instTcpSend.REQ := true;


                        IF ((#instTcpSend.DONE)
                            AND (#instTcpSend.BUSY = 0))
                        THEN
                            #instTcpSend.REQ := false;
                            IF (#mqttParam.publishFlag.qualityOfService > 0)
                            THEN
                                #statPacketIDAck := #statPacketID;
                                #statStateMQTTinternal := #MQTT_PUBACK;
                            ELSE
                                //QoS = 0; finish here
                                #published := true;
                                #busy := false;
                                #statNewDataRcv := false;
                                IF NOT #statKeepAliveOff
                                THEN
                                    #statTriggerKeepAlive := true;
                                END_IF;

                                #statStateMQTTinternal := #IDLE;
                            END_IF;
                        ELSIF #instTcpSend.ERROR
                        THEN
                            #statusID := #MQTT_PUBLISH;
                            #instTcpSend.REQ := false;
                            #statStateMQTT := #MQTT_ERROR;
                            #status := #instTcpSend.STATUS;
                        END_IF;
                    #MQTT_PUBACK:
                        IF #statNewDataRcv THEN
                            IF ((#statRcvBuffer[1] AND b#16#f0) = #MQTT_MSG_TYPE_PUBACK)
                                OR
                                ((#statRcvBuffer[1] AND b#16#f0) = INT_TO_WORD(#MQTT_MSG_TYPE_PUBREC))
                            THEN
                                IF
                                    (#statRcvBuffer[3] = #statPacketIDAck.%B1)
                                    AND
                                    (#statRcvBuffer[4] = #statPacketIDAck.%B0)
                                THEN
                                    IF (#mqttParam.publishFlag.qualityOfService = 1)
                                    THEN
                                        //QoS = 1; finish here
                                        #statStateMQTTinternal := #MQTT_IDLE;
                                        #published := true;
                                        #busy := false;
                                        #statNewDataRcv := false;
                                        //Re-Activate Kepp Alive Timer
                                        IF NOT #statKeepAliveOff
                                        THEN
                                            #statTriggerKeepAlive := true;
                                        END_IF;

                                        #statStateMQTTinternal := #IDLE;
                                    ELSE
                                        #statStateMQTTinternal := #MQTT_PUBREL;
                                    END_IF;
                                ELSE
                                    #statNewDataRcv := false;
                                END_IF;
                            ELSE
                                #statStateMQTT := #MQTT_ERROR;
                                #statusID := #MQTT_PUBACK;
                            END_IF;
                        END_IF;
                    #MQTT_PUBREL:
                        //fixed Header
                        #statSendBuffer[1] := 16#62;
                        #statSendBuffer[2] := 2;
                        //Variable Header
                        #statSendBuffer[3] := #statPacketID.%B1;
                        #statSendBuffer[4] := #statPacketID.%B0;
                        #instTcpSend.LEN := INT_TO_UDINT(4);
                        #instTcpSend.REQ := true;

                        IF ((#instTcpSend.DONE)
                            AND (#instTcpSend.BUSY = 0))
                        THEN
                            #instTcpSend.REQ := false;
                            #statPacketIDAck := #statPacketID;
                            #statStateMQTTinternal := #MQTT_PUBCOMP;

                        ELSIF #instTcpSend.ERROR
                        THEN
                            #statusID := #MQTT_PUBREL;
                            #instTcpSend.REQ := false;
                            #statStateMQTT := #MQTT_ERROR;
                            #status := #instTcpSend.STATUS;
                        END_IF;
                    #MQTT_PUBCOMP:
                        IF #statNewDataRcv THEN
                            IF ((#statRcvBuffer[1] AND b#16#f0) = #MQTT_MSG_TYPE_PUBCOM)
                            THEN
                                IF
                                    (#statRcvBuffer[3] = #statPacketIDAck.%B1)
                                    AND
                                    (#statRcvBuffer[4] = #statPacketIDAck.%B0)
                                THEN
                                    //QoS = 2; finish here
                                    #statStateMQTTinternal := #MQTT_IDLE;
                                    #published := true;
                                    #busy := false;
                                    #statNewDataRcv := false;
                                    //Re-Activate Kepp Alive Timer
                                    IF NOT #statKeepAliveOff
                                    THEN
                                        #statTriggerKeepAlive := true;
                                    END_IF;

                                    #statStateMQTTinternal := #IDLE;
                                ELSE
                                    #statStateMQTT := #MQTT_ERROR;
                                    #statusID := #MQTT_PUBCOMP;
                                END_IF;
                            END_IF;
                        END_IF;
                    #MQTT_PING:

                        #busy := true;
                        //Build fixed Header
                        //Message Type
                        #statSendBuffer[1] := INT_TO_BYTE(#MQTT_MSG_TYPE_PING);
                        //Remaining Lenght (must be O)
                        #statSendBuffer[2] := 0;
                        #instTcpSend.REQ := true;
                        #instTcpSend.LEN := 2;

                        IF ((#instTcpSend.DONE)
                            AND (#instTcpSend.BUSY = 0))
                        THEN
                            #instTcpSend.REQ := false;
                            #statStateMQTTinternal := #MQTT_PINGRESP;
                        ELSIF #instTcpSend.ERROR
                        THEN
                            #statusID := #MQTT_PING;
                            #instTcpSend.REQ := false;
                            #statStateMQTT := #MQTT_ERROR;
                            #status := #instTcpSend.STATUS;
                        END_IF;
                    #MQTT_PINGRESP:
                        IF #statNewDataRcv
                        THEN
                            IF ((#statRcvBuffer[1] AND b#16#f0) = #MQTT_MSG_TYPE_PINGRESP)
                            THEN
                                #busy := false;
                                #statNewDataRcv := false;
                                #statTriggerKeepAlive := true;
                                #statStateMQTTinternal := #IDLE;
                            END_IF;
                        ELSE
                            #statNewDataRcv := false;
                        END_IF;

                END_CASE;
           #MQTT_DISCONNECT:
           #busy := 0;
           //Build fixed Header
           //Message Type
           #statSendBuffer[1] := INT_TO_BYTE(#MQTT_MSG_TYPE_DISCONNECT);
           //Remaining Lenght (must be O)
           #statSendBuffer[2] := 0;
           #instTcpSend.REQ := true;
           #instTcpSend.LEN := 2;

           IF ((#instTcpSend.DONE)
               AND (#instTcpSend.BUSY = 0))
           THEN
               IF NOT #enable THEN
                   #statStateTCP := #TCP_DISCONNECT;
               END_IF;
               #instTcpSend.REQ := false;
               #statStateMQTT := #MQTT_DISCONNECTED;
               #statStateMQTTinternal := #IDLE;
           ELSIF #instTcpSend.ERROR
           THEN
               IF NOT #enable THEN
                   #statStateTCP := #TCP_DISCONNECT;
               END_IF;
               #statusID := #MQTT_DISCONNECT;
               #instTcpSend.REQ := false;
               #statStateMQTT := #MQTT_ERROR;
               #status := #instTcpSend.STATUS;
           END_IF;
               #MQTT_ERROR:

               REGION Errorhandling MQTT
                   #error := true;
                   #busy := false;
                   #statStateMQTTinternal := #IDLE;
                   #statTriggerKeepAlive := 0;
                   #statKeepAliveOff := false;
                 CASE #statusID OF
                     #MQTT_CONNECT_FLAG_CHECK:
                         #mqttEstablished := false;
                         #statStateMQTT := #MQTT_DISCONNECTED;
                         ;
                     #MQTT_CONNECT:
                         #mqttEstablished := false;
                         #status := #instTcpSend.STATUS;   ;
                         #statStateMQTT := #MQTT_DISCONNECTED;
                       #MQTT_CONNACK:
                           #mqttEstablished := false;
                           #status := #statRcvBuffer[4];
                           #statStateMQTT := #MQTT_DISCONNECTED;
                       #MQTT_PUBLISH:
                               #published := false;
                               #statStateMQTT := #MQTT_CONNECTED;
                               #MQTT_PUBACK,#MQTT_PUBCOMP,#MQTT_PUBREL:
                           #published := false;
                           #status :=#MQTT_ERROR_PACKETID;
                           #statStateMQTT := #MQTT_CONNECTED;
                       #MQTT_PINGRESP:;
                           #MQTT_PING:;
                       #MQTT_DISCONNECT:
                           #mqttEstablished := false;
                          ;
                       ELSE
                           ;
                   END_CASE;
              END_REGION
               ;



       END_CASE
       ;
END_FUNCTION_BLOCK